Staubli VAL3: Vereinzeln.pgx

program Vereinzeln()
  local mdesc mDesc
  local bool error
  local num i
begin


  while true

    // Vereinzelt die Objekte


    wait(bNewData)

    // Wenn wir nicht vereinzeln heben wir Obj auf und setzen diese ab
    if bVereinzeln
      logMsg("Vereinzeln startet ")

      pVereinzeln.trsf.x = nX
      pVereinzeln.trsf.y = nY
      pVereinzeln.trsf.rz = nAngle


      //logMsg("nAngle ****************** " + toString("0.4", nAngle))
      //logMsg("nData ****************** " + toString("0.4", nData[4] ))
      close(tGreiferM)
      // Fahre über Punkt Vereinzeln --> irgenwie
      movej(appro(pVereinzeln, trApro), tGreiferM, mUsedSpeed)


      movej(pVereinzeln, tGreiferM, mVereinzeln)

      // Fahre linear trVer voraus
      pVereinzeln.trsf.x =  pVereinzeln.trsf.x +  100 * cos(-nData[4])
      pVereinzeln.trsf.y =  pVereinzeln.trsf.y +  100 * sin(-nData[4])

      movej(pVereinzeln,tGreiferM, mVereinzeln)
      // fahre vom letzten POSE appro(pVereinzeln,trVer) --> zur neuen oberhalb, --> trApro

      // Überprüft ob die EndPOSE erreichbar ist sonst verändere den Winkel
      i = 0
      error = false
      while !pointToJoint(tGreiferM,jHome,appro(pVereinzeln, trApro),jEmpty) and  error == false
        pVereinzeln.trsf.rz = pVereinzeln.trsf.rz + 5
        i = i +1
        if i > 100
          error = true
        endIf
      endWhile

      if !error
        movej(appro(pVereinzeln, trApro), tGreiferM, mVereinzeln)
      endIf





      //logMsg("Objekt vereinzelt")

      // Return Value
      bNewData = false
      bReady = true


    endIf








  endWhile

end
